Staubli VAL3: getGeometricMean.pgx

public program getGeometricMean(num& x_nInput[], num& x_nMean)
  local num l_nCount
  local num l_nProd
begin

  l_nProd = 1

  for l_nCount = 0 to size(x_nInput)-1
    l_nProd = l_nProd * x_nInput[l_nCount]
  endFor
  ? l_nProd
  x_nMean = power(l_nProd,1/size(x_nInput))

end
